FUNCTION_BLOCK POSTGRE_DB_FETCH_JSON_TIMESERIES
  {SET_ATTRIBUTE(OpcUa, POINT.ENDPOINT)}
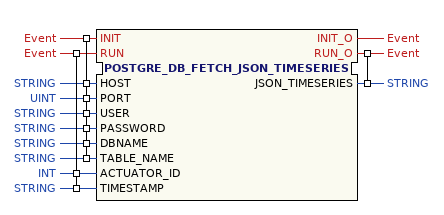
  EVENT_INPUT
    INIT WITH HOST, PORT, USER, PASSWORD, DBNAME, TABLE_NAME;
    RUN WITH ACTUATOR_ID, TIMESTAMP;
  END_EVENT
  EVENT_OUTPUT
    INIT_O;
    RUN_O WITH JSON_TIMESERIES;
  END_EVENT
  VAR_INPUT
    HOST : STRING; {SET_ATTRIBUTE(OpcUa, Constant)}
    PORT : UINT; {SET_ATTRIBUTE(OpcUa, Constant)}
    USER : STRING; {SET_ATTRIBUTE(OpcUa, Constant)}
    PASSWORD : STRING; {SET_ATTRIBUTE(OpcUa, Constant)}
    DBNAME : STRING; {SET_ATTRIBUTE(OpcUa, Constant)}
    TABLE_NAME : STRING; {SET_ATTRIBUTE(OpcUa, Constant)}
    ACTUATOR_ID : INT; {SET_ATTRIBUTE(OpcUa, Constant)}
    TIMESTAMP : STRING; {SET_ATTRIBUTE(OpcUa, Constant)}
  END_VAR
  VAR_OUTPUT
    JSON_TIMESERIES : STRING; {SET_ATTRIBUTE(OpcUa, Variable.RUN)}
  END_VAR
END_FUNCTION_BLOCK
